# EPICS substitutions: db/Beckhoff_2XXX/ecmcEP2308.substitutions
# binary outputs
file "ecmc_binaryOutput-chX.template"{
  pattern {CH_ID}
          {01   }
          {02   }
          {03   }
          {04   }
}

# binary inputs
file "ecmc_binaryInput-chX.template"{
  pattern {CH_ID}
          {01   }
          {02   }
          {03   }
          {04   }
}
